(* A flashing beacon made from two timers. It runs by itself as soon as the simulator starts. Force Enable FALSE to stop it. *)

PROGRAM P3_Flasher
  VAR
    Enable : BOOL := TRUE; (* Beacon enabled *)
    OnTimer : TON; (* Times the lit half of the cycle *)
    OffTimer : TON; (* Times the dark half of the cycle *)
    OnDone : BOOL; (* Lit half finished *)
    OffDone : BOOL; (* Dark half finished *)
    Beacon : BOOL; (* Flashing beacon: 0.5 s on, 0.5 s off *)
  END_VAR

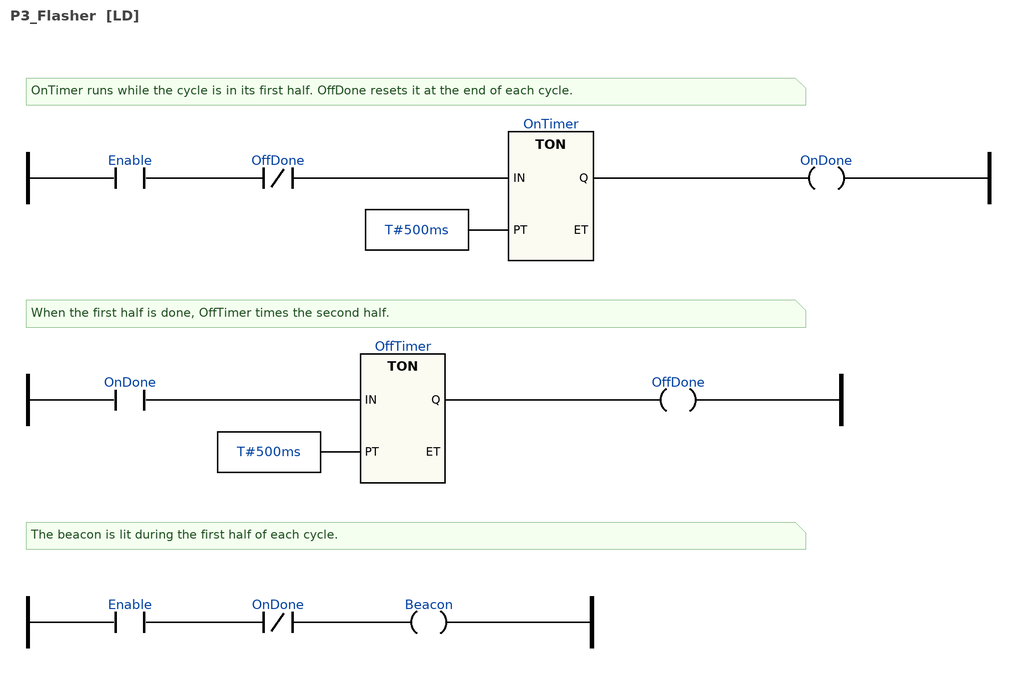
(* LD diagram, written out as Structured Text *)
(* OnTimer runs while the cycle is in its first half. OffDone resets it at the end of each cycle. *)
OnTimer(IN := Enable AND NOT OffDone, PT := T#500ms);
OnDone := OnTimer.Q;
(* When the first half is done, OffTimer times the second half. *)
OffTimer(IN := OnDone, PT := T#500ms);
OffDone := OffTimer.Q;
(* The beacon is lit during the first half of each cycle. *)
Beacon := Enable AND NOT OnDone;
END_PROGRAM
